(* Schneider Machine Expert - Basic project _M5.4 Schedule Block Gral, file version 2.6.0.0 *)
(* CompanyInformations: Name=Schneider Electric, PhoneNumber=+44 870 608 8608, Street=Stafford Park 5, City=Telford, ZipCode=TF3 3BL, Country=United Kingdom, WebSite=se.com/uk *)
(* ProjectInformations: Name=M221 - BASIC FUNCTIONs, Description=In this demo project the following function blocks are used:
•RTC ( only Write mode in simulation) *)
(* UserInformations: LastName=Ahumada, FirstName=Leandro, PhoneNumber=+44 870 608 8608, Email=leandro.ahumada@se.com, Street=Stafford Park 5, City=Telford, ZipCode=TF3 3BL, Country=United Kingdom *)

HARDWARE
  Cpu 0: TM221CE24R
  EthernetConfiguration: NetworkName=M221, IpAllocationMode=FixedAddress, IpAddress=192.168.1.221, SubnetMask=255.255.255.0
  SerialLineConfiguration: Baud=Baud19200, Parity=ParityEven, DataBits=DataBits8, StopBits=StopBits1, PhysicalMedium=PhysicalMediumRs485, TransmissionMode=TransmissionModeModbusRtu, SlaveId=1, Addressing=SlaveAddressing
  MastTask: UsePeriodScanMode=false, PeriodScan=100
  FastTask: Period=255
  CpuBehavior: StartingMode=StartAsPreviousState, AutoSaveRamOnEeprom=true, WatchdogPeriod=250

SYMBOLS  (address, symbol, comment, settings)
  %M22      CFG_SCH_MONDAY
  %M23      CFG_SCH_TUESDAY
  %M24      CFG_SCH_WEDNESDAY
  %M25      CFG_SCH_THURSDAY
  %M26      CFG_SCH_FRIDAY
  %M27      CFG_SCH_SATURDAY
  %M28      CFG_SCH_SUNDAY
  %M80      PET_RTC_ENABLE  "At state 1, the RD and WR input values are read continuously to determine the action to take."
  %M81      PET_RTC_READ  "RD = 1 and WR = 0. Read the RTC value."
  %M82      PET_RTC_WRITE  "RD = 0 and WR = 1. When the rising edge of WR is detected, update the RTC using the object values specified in the RTC parameter"
  %M83      IND_RTC_DONE  "Set to 1 when the RTC is successfully read from or written to."
  %M84      IND_RTC_ERROR  "The ErrorId output object indicates the cause of the error."
  %S50      SB_RTCUPDATE  "Set to 1, this bit allows to update the date and time"
  %SW50     SW_RTCSEC  "RTC Function: contains in BCD 00SS Seconds"
  %SW51     SW_RTCHHMM  "RTC Function: contains in BCD HHMM: hour and minute"
  %SW52     SW_RTCMMDD  "RTC Function: contains in BCD MMDD: month and day"
  %SW53     SW_RTCCCYY  "RTC Function: contains in BCD CCYY: century and year"
  %MW0      IND_RTC_SYSTEM_YEAR  "Using the %SW53"
  %MW1      IND_RTC_SYSTEM_DAY  "Using the %SW52 + SHL + BTI"
  %MW2      IND_RTC_SYSTEM_MONTH  "Using the %SW52 + SHL + BTI"
  %MW3      IND_RTC_SYSTEM_SEC  "Using the %SW50"
  %MW4      IND_RTC_SYSTEM_MIN  "Using the %SW51+ SHL + BTI"
  %MW5      IND_RTC_SYSTEM_HOUR  "Using the %SW51 + SHL + BTI"
  %MW6      CFG_RT_SYSTEM_YEAR
  %MW7      CFG_RTC_SYSTEM_DAY
  %MW8      CFG_RTC_SYSTEM_MONTH
  %MW9      CFG_RTC_SYSTEM_SEC
  %MW10     CFG_RTC_SYSTEM_MIN
  %MW11     CFG_RTC_SYSTEM_HOUR
  %MW20     CFG_SCH_STARTDAY  "Config. - Schedule - Start day"
  %MW21     CFG_SCH_STARTMONTH  "Config. - Schedule - Start month"
  %MW22     CFG_SCH_STARTHOUR  "Config. - Schedule - Start hour"
  %MW23     CFG_SCH_STARTMIN  "Config. - Schedule - Start min"
  %MW24     CFG_SCH_ENDDAY  "Config. - Schedule - End day"
  %MW25     CFG_SCH_ENDMONTH  "Config. - Schedule - End month"
  %MW26     CFG_SCH_ENDHOUR  "Config. - Schedule - End hour"
  %MW27     CFG_SCH_ENDMIN
  %MW28     CFG_SCH_DOW  "Config. - Schedule - Day of week"
  %MW41     IND_RTC_IDERROR
  %MW42     IND_RTC_ACTUAL_DAY
  %MW43     IND_RTC_ACTUAL_MONTH
  %MW44     IND_RTC_ACTUAL_YEAR
  %MW45     IND_RTC_ACTUAL_HH
  %MW46     IND_RTC_ACTUAL_MM
  %MW47     IND_RTC_ACTUAL_SS
  %MW48     IND_RTC_ACTUAL_DAYOFWEEK
  %MW50     IND_RTC_WRITE_DAY
  %MW51     IND_RTC_WRITE_MONTH
  %MW52     IND_RTC_WRITE_YEAR
  %MW53     IND_RTC_WRITE_HH
  %MW54     IND_RTC_WRITE_MM
  %MW55     IND_RTC_WRITE_SS
  %SCH0       [Configured=true, OutputBit=%M1, StartDate=2012-01-01T00:00:00, EndDate=2012-01-01T00:00:00]
  %RTC0     INST_RTC  [Day(Value(int=24)), Month(Value(int=12)), Year(Value(int=2019)), Hours(Value(int=0)), Minutes(Value(int=0)), Seconds(Value(int=0))]

POU PRG_RTC
  (* SectionNumber=1 *)

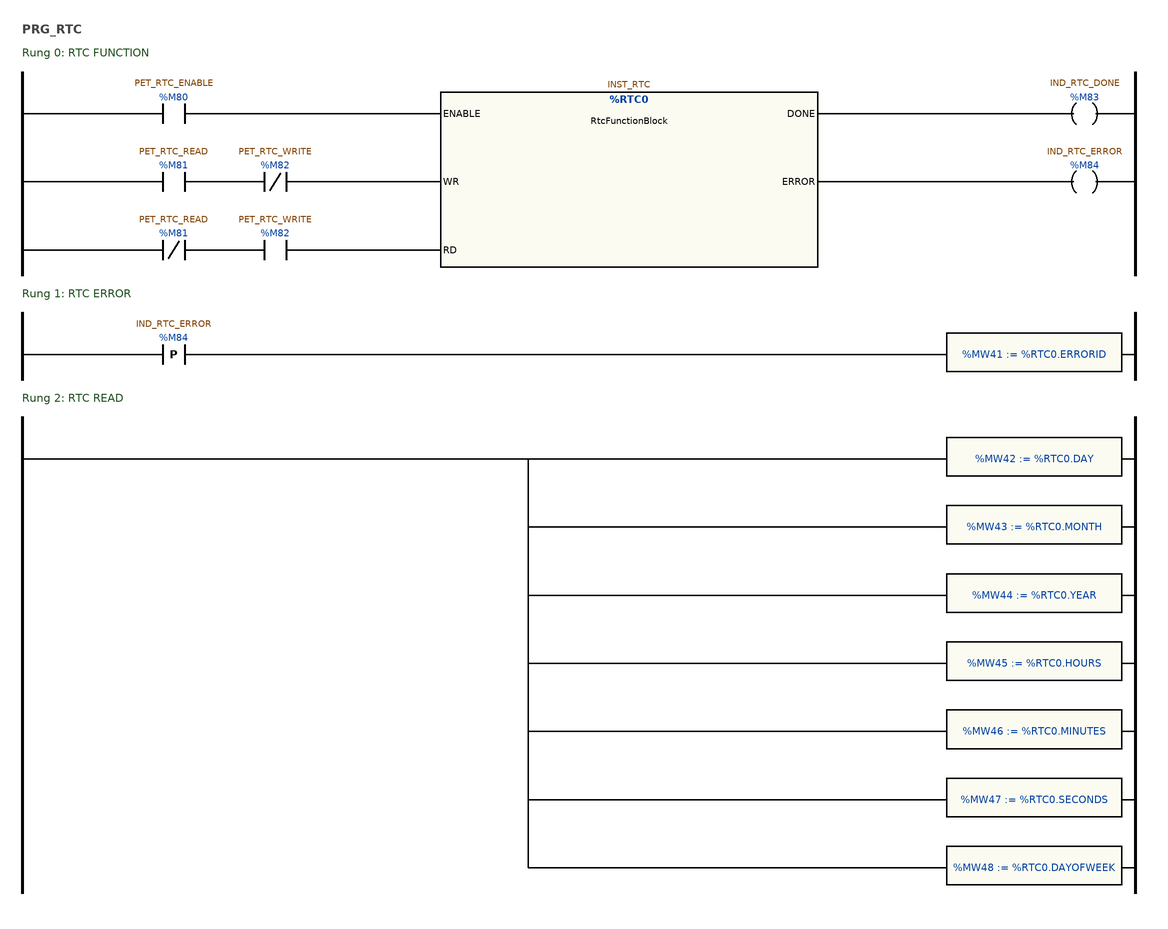

// Rung 0: RTC FUNCTION
  BLK %RTC0               (* INST_RTC *)
  LD %M80                 (* PET_RTC_ENABLE *)
  ENABLE
  LD %M81                 (* PET_RTC_READ *)
  ANDN %M82               (* PET_RTC_WRITE *)
  WR
  LDN %M81                (* PET_RTC_READ *)
  AND %M82                (* PET_RTC_WRITE *)
  RD
  OUT_BLK
  LD DONE
  ST %M83                 (* IND_RTC_DONE *)
  LD ERROR
  ST %M84                 (* IND_RTC_ERROR *)
  END_BLK
  // as ST:
  //   INST_RTC(ENABLE := PET_RTC_ENABLE, WR := PET_RTC_READ AND NOT PET_RTC_WRITE, RD := NOT PET_RTC_READ AND PET_RTC_WRITE);
  //   IND_RTC_DONE := INST_RTC.DONE;
  //   IND_RTC_ERROR := INST_RTC.ERROR;

// Rung 1: RTC ERROR
  LDR %M84                (* IND_RTC_ERROR *)
  [ %MW41 := %RTC0.ERRORID ](* IND_RTC_IDERROR, INST_RTC *)
  // as ST:
  //   IF RISING(IND_RTC_ERROR) THEN IND_RTC_IDERROR := INST_RTC.ERRORID; END_IF;

// Rung 2: RTC READ
  LD 1
  [ %MW42 := %RTC0.DAY ]  (* IND_RTC_ACTUAL_DAY, INST_RTC *)
  [ %MW43 := %RTC0.MONTH ](* IND_RTC_ACTUAL_MONTH, INST_RTC *)
  [ %MW44 := %RTC0.YEAR ] (* IND_RTC_ACTUAL_YEAR, INST_RTC *)
  [ %MW45 := %RTC0.HOURS ](* IND_RTC_ACTUAL_HH, INST_RTC *)
  [ %MW46 := %RTC0.MINUTES ](* IND_RTC_ACTUAL_MM, INST_RTC *)
  [ %MW47 := %RTC0.SECONDS ](* IND_RTC_ACTUAL_SS, INST_RTC *)
  [ %MW48 := %RTC0.DAYOFWEEK ](* IND_RTC_ACTUAL_DAYOFWEEK, INST_RTC *)
  // as ST:
  //   IND_RTC_ACTUAL_DAY := INST_RTC.DAY;
  //   IND_RTC_ACTUAL_MONTH := INST_RTC.MONTH;
  //   IND_RTC_ACTUAL_YEAR := INST_RTC.YEAR;
  //   IND_RTC_ACTUAL_HH := INST_RTC.HOURS;
  //   IND_RTC_ACTUAL_MM := INST_RTC.MINUTES;
  //   IND_RTC_ACTUAL_SS := INST_RTC.SECONDS;
  //   IND_RTC_ACTUAL_DAYOFWEEK := INST_RTC.DAYOFWEEK;

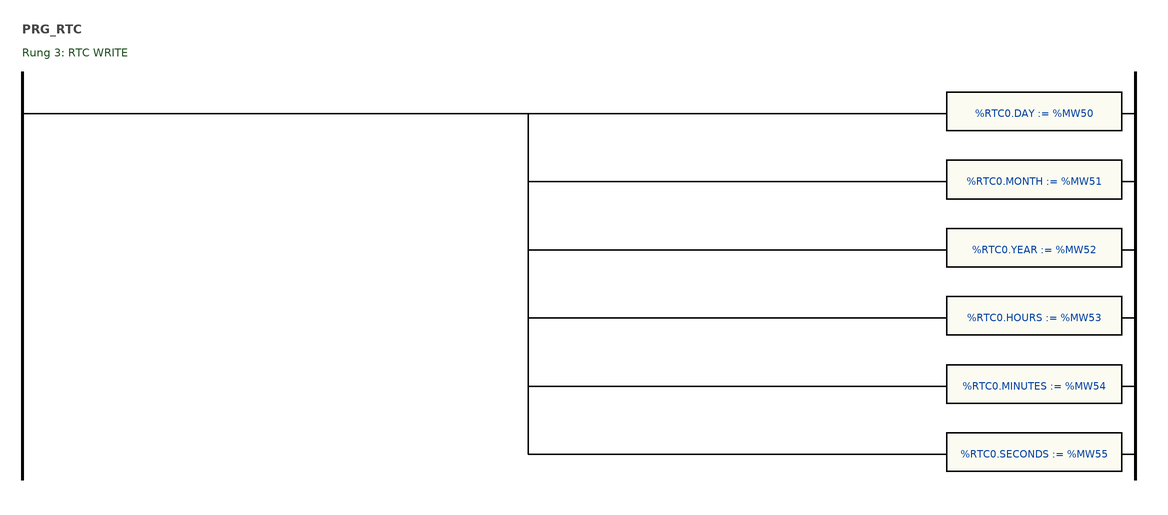

// Rung 3: RTC WRITE
  LD 1
  [ %RTC0.DAY := %MW50 ]  (* INST_RTC, IND_RTC_WRITE_DAY *)
  [ %RTC0.MONTH := %MW51 ](* INST_RTC, IND_RTC_WRITE_MONTH *)
  [ %RTC0.YEAR := %MW52 ] (* INST_RTC, IND_RTC_WRITE_YEAR *)
  [ %RTC0.HOURS := %MW53 ](* INST_RTC, IND_RTC_WRITE_HH *)
  [ %RTC0.MINUTES := %MW54 ](* INST_RTC, IND_RTC_WRITE_MM *)
  [ %RTC0.SECONDS := %MW55 ](* INST_RTC, IND_RTC_WRITE_SS *)
  // as ST:
  //   INST_RTC.DAY := IND_RTC_WRITE_DAY;
  //   INST_RTC.MONTH := IND_RTC_WRITE_MONTH;
  //   INST_RTC.YEAR := IND_RTC_WRITE_YEAR;
  //   INST_RTC.HOURS := IND_RTC_WRITE_HH;
  //   INST_RTC.MINUTES := IND_RTC_WRITE_MM;
  //   INST_RTC.SECONDS := IND_RTC_WRITE_SS;

POU PRG_RTC_System
  (* SectionNumber=2 *)

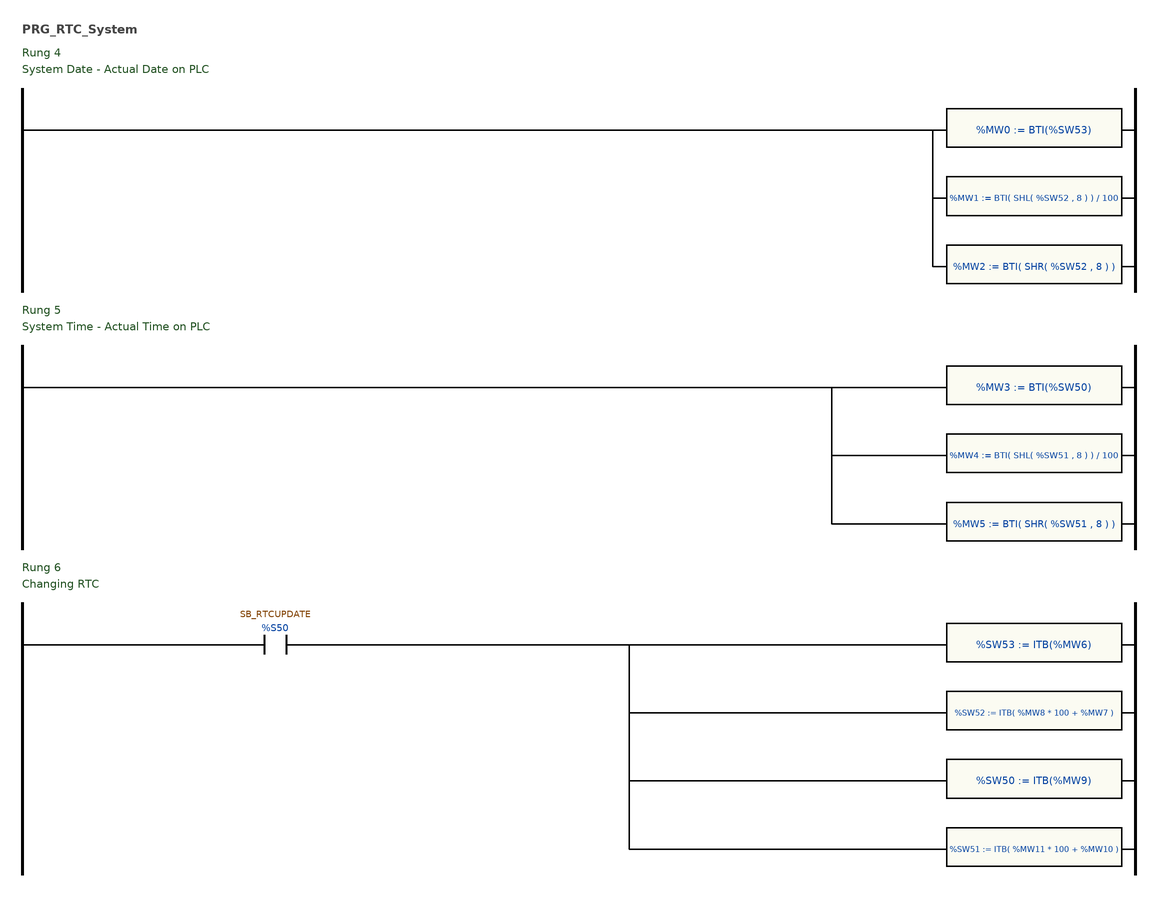

// Rung 4
// System Date - Actual Date on PLC
  LD 1
  [ %MW0 := BTI ( %SW53 ) ](* IND_RTC_SYSTEM_YEAR, SW_RTCCCYY *)
  [ %MW1 := BTI ( SHL ( %SW52 , 8 ) ) / 100 ](* IND_RTC_SYSTEM_DAY, SW_RTCMMDD *)
  [ %MW2 := BTI ( SHR ( %SW52 , 8 ) ) ](* IND_RTC_SYSTEM_MONTH, SW_RTCMMDD *)
  // as ST:
  //   IND_RTC_SYSTEM_YEAR := BTI ( SW_RTCCCYY );
  //   IND_RTC_SYSTEM_DAY := BTI ( SHL ( SW_RTCMMDD , 8 ) ) / 100;
  //   IND_RTC_SYSTEM_MONTH := BTI ( SHR ( SW_RTCMMDD , 8 ) );

// Rung 5
// System Time - Actual Time on PLC
  LD 1
  [ %MW3 := BTI ( %SW50 ) ](* IND_RTC_SYSTEM_SEC, SW_RTCSEC *)
  [ %MW4 := BTI ( SHL ( %SW51 , 8 ) ) / 100 ](* IND_RTC_SYSTEM_MIN, SW_RTCHHMM *)
  [ %MW5 := BTI ( SHR ( %SW51 , 8 ) ) ](* IND_RTC_SYSTEM_HOUR, SW_RTCHHMM *)
  // as ST:
  //   IND_RTC_SYSTEM_SEC := BTI ( SW_RTCSEC );
  //   IND_RTC_SYSTEM_MIN := BTI ( SHL ( SW_RTCHHMM , 8 ) ) / 100;
  //   IND_RTC_SYSTEM_HOUR := BTI ( SHR ( SW_RTCHHMM , 8 ) );

// Rung 6
// Changing RTC
  LD %S50                 (* SB_RTCUPDATE *)
  [ %SW53 := ITB ( %MW6 ) ](* SW_RTCCCYY, CFG_RT_SYSTEM_YEAR *)
  [ %SW52 := ITB ( %MW8 * 100 + %MW7 ) ](* SW_RTCMMDD, CFG_RTC_SYSTEM_MONTH, CFG_RTC_SYSTEM_DAY *)
  [ %SW50 := ITB ( %MW9 ) ](* SW_RTCSEC, CFG_RTC_SYSTEM_SEC *)
  [ %SW51 := ITB ( %MW11 * 100 + %MW10 ) ](* SW_RTCHHMM, CFG_RTC_SYSTEM_HOUR, CFG_RTC_SYSTEM_MIN *)
  // as ST:
  //   IF SB_RTCUPDATE THEN SW_RTCCCYY := ITB ( CFG_RT_SYSTEM_YEAR ); END_IF;
  //   IF SB_RTCUPDATE THEN SW_RTCMMDD := ITB ( CFG_RTC_SYSTEM_MONTH * 100 + CFG_RTC_SYSTEM_DAY ); END_IF;
  //   IF SB_RTCUPDATE THEN SW_RTCSEC := ITB ( CFG_RTC_SYSTEM_SEC ); END_IF;
  //   IF SB_RTCUPDATE THEN SW_RTCHHMM := ITB ( CFG_RTC_SYSTEM_HOUR * 100 + CFG_RTC_SYSTEM_MIN ); END_IF;

POU PRG_SCHEDULE
  (* SectionNumber=3 *)

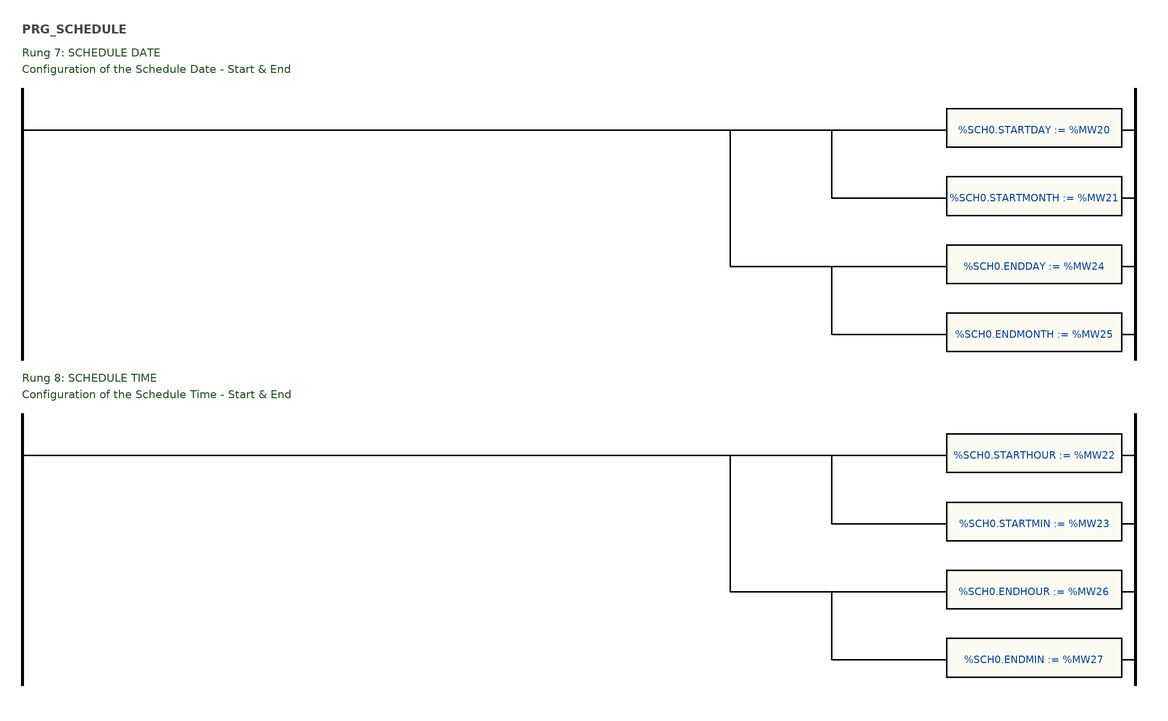

// Rung 7: SCHEDULE DATE
// Configuration of the Schedule Date - Start & End
  LD 1
  [ %SCH0.STARTDAY := %MW20 ](* CFG_SCH_STARTDAY *)
  [ %SCH0.STARTMONTH := %MW21 ](* CFG_SCH_STARTMONTH *)
  [ %SCH0.ENDDAY := %MW24 ](* CFG_SCH_ENDDAY *)
  [ %SCH0.ENDMONTH := %MW25 ](* CFG_SCH_ENDMONTH *)
  // as ST:
  //   %SCH0.STARTDAY := CFG_SCH_STARTDAY;
  //   %SCH0.STARTMONTH := CFG_SCH_STARTMONTH;
  //   %SCH0.ENDDAY := CFG_SCH_ENDDAY;
  //   %SCH0.ENDMONTH := CFG_SCH_ENDMONTH;

// Rung 8: SCHEDULE TIME
// Configuration of the Schedule Time - Start & End
  LD 1
  [ %SCH0.STARTHOUR := %MW22 ](* CFG_SCH_STARTHOUR *)
  [ %SCH0.STARTMIN := %MW23 ](* CFG_SCH_STARTMIN *)
  [ %SCH0.ENDHOUR := %MW26 ](* CFG_SCH_ENDHOUR *)
  [ %SCH0.ENDMIN := %MW27 ](* CFG_SCH_ENDMIN *)
  // as ST:
  //   %SCH0.STARTHOUR := CFG_SCH_STARTHOUR;
  //   %SCH0.STARTMIN := CFG_SCH_STARTMIN;
  //   %SCH0.ENDHOUR := CFG_SCH_ENDHOUR;
  //   %SCH0.ENDMIN := CFG_SCH_ENDMIN;

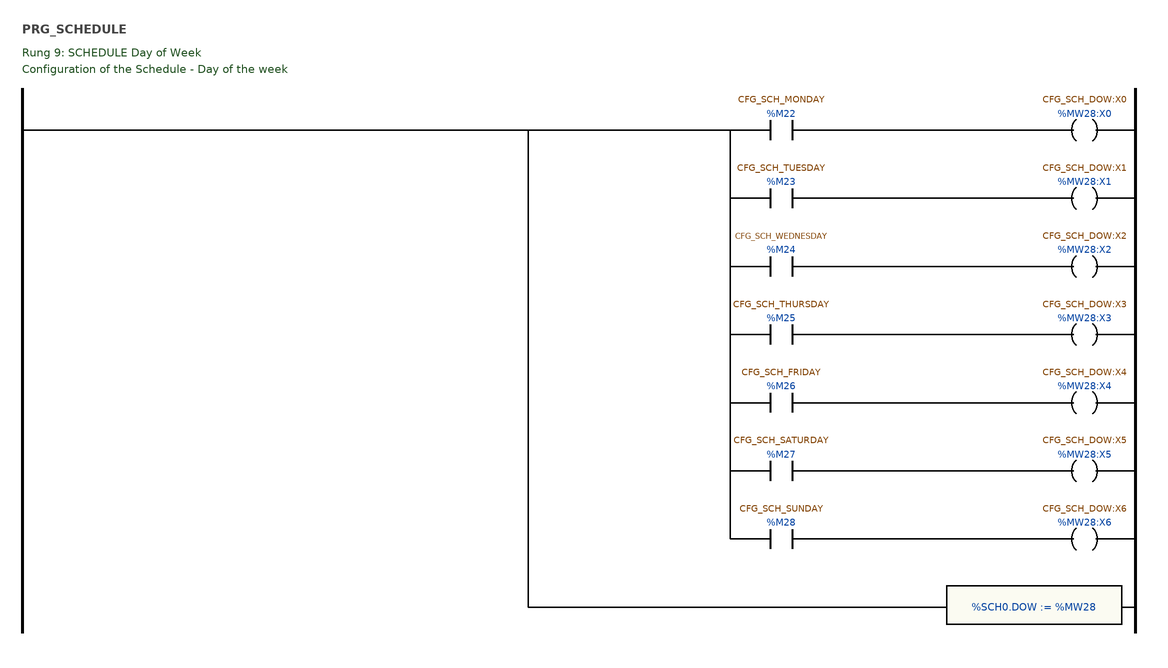

// Rung 9: SCHEDULE Day of Week
// Configuration of the Schedule - Day of the week
  LD 1
  MPS
  AND %M22                (* CFG_SCH_MONDAY *)
  ST %MW28:X0             (* CFG_SCH_DOW *)
  MRD
  AND %M23                (* CFG_SCH_TUESDAY *)
  ST %MW28:X1             (* CFG_SCH_DOW *)
  MRD
  AND %M24                (* CFG_SCH_WEDNESDAY *)
  ST %MW28:X2             (* CFG_SCH_DOW *)
  MRD
  AND %M25                (* CFG_SCH_THURSDAY *)
  ST %MW28:X3             (* CFG_SCH_DOW *)
  MRD
  AND %M26                (* CFG_SCH_FRIDAY *)
  ST %MW28:X4             (* CFG_SCH_DOW *)
  MRD
  AND %M27                (* CFG_SCH_SATURDAY *)
  ST %MW28:X5             (* CFG_SCH_DOW *)
  MRD
  AND %M28                (* CFG_SCH_SUNDAY *)
  ST %MW28:X6             (* CFG_SCH_DOW *)
  MPP
  [ %SCH0.DOW := %MW28 ]  (* CFG_SCH_DOW *)
  // as ST:
  //   CFG_SCH_DOW:X0 := CFG_SCH_MONDAY;
  //   CFG_SCH_DOW:X1 := CFG_SCH_TUESDAY;
  //   CFG_SCH_DOW:X2 := CFG_SCH_WEDNESDAY;
  //   CFG_SCH_DOW:X3 := CFG_SCH_THURSDAY;
  //   CFG_SCH_DOW:X4 := CFG_SCH_FRIDAY;
  //   CFG_SCH_DOW:X5 := CFG_SCH_SATURDAY;
  //   CFG_SCH_DOW:X6 := CFG_SCH_SUNDAY;
  //   %SCH0.DOW := CFG_SCH_DOW;
